INTERFACE I_InSafetyGroup EXTENDS I_Base

PROPERTY SafetyGroup : I_TaskResult
SET
END_SET
END_PROPERTY

END_INTERFACE

(* stored: Version 1.1.0.1, ProductVersion 3.1.4026.18
   Itf I_InSafetyGroup: Id {103af291-27bd-4f2e-84a7-37f9e3654eff}
   Property SafetyGroup: Id {0b114d3b-7457-419e-850b-91910b1e8c2e}
   Set Set: Id {4f569d64-cc5b-453b-87fc-c8cef5482f49} *)
